// TIA Portal V20 export
TYPE "typeSequenceControlNodeHomeCheck"
// stored: Namespace Unit1.Em7
   STRUCT
      liftDownPartNoDetect : Bool;
      liftDownPartDetect : Bool;
      liftUp : Bool;
   END_STRUCT;
END_TYPE
